Staubli VAL3: page.pgx

public program page(string& menuname[], num index)
// set all the page in italian PALLET
begin
  //
  //  PAGE
  //
  // PALLET PAGE
  if index>=10 and index<=19
    title("< Gestione Pallet >")
  endIf
  // PALLET VIEW PAGE
  if index>=100 and index<=109
    title("< Configurazione Pallet >")
  endIf
  switch index
    //
    // PALLET
    //
    // Integrator programmer
    case 10,11
      menuname="Vedi Programma,Modifica,,,Assistente,Inizializza,Indietro,Avanti"
    break
    // On Cycle
    case 13,14
      menuname="Vedi Programma,Modifica,,,Assistente,Inizializza,Indietro,Avanti"
    break
    // VIEW PALLET
    case 100,101,102,103,104,105
      menuname="Inizializza,,,,,Zero,Indietro,Avanti"
    break
  endSwitch
end
